// TwinCAT 3 PLC project PLC1
// ProgramVersion: 3.1.4026.16
// libraries:
//   Tc2_Standard, * (Beckhoff Automation GmbH)
//   Tc2_System, * (Beckhoff Automation GmbH)
// project tree:
//   DUTs/ YOLO_OBJECT_DETECTION.TcDUT
//   / PlcTask.TcTTO
//   POUs/ CountAndKeepValidDetections.TcPOU, MAIN.TcPOU, NonMaximumSuppression.TcPOU, SortDetectionsByConfidence.TcPOU
// real-time tasks:
//   TASK PlcTask: cycle T#10ms, priority 20, ADS port 350

CONFIGURATION PLC1
    RESOURCE PLC ON TwinCAT3
        TASK PlcTask(INTERVAL := T#10ms, PRIORITY := 20);
        PROGRAM MAIN WITH PlcTask : MAIN;
    END_RESOURCE
END_CONFIGURATION

// ---- DUTs/YOLO_OBJECT_DETECTION.TcDUT
TYPE YOLO_OBJECT_DETECTION :
STRUCT
	x_center_px 	: REAL;
    y_center_px 	: REAL;
    width_px    	: REAL;
    height_px   	: REAL;
    confidence  	: REAL;
	nTopLeftX       : REAL;
    nTopLeftY       : REAL;
    nBottomRightX   : REAL;
    nBottomRightY   : REAL;
    valid       	: BOOL; // For NMS marking
END_STRUCT
END_TYPE

// ---- POUs/MAIN.TcPOU
PROGRAM MAIN
VAR
	arrDetections : ARRAY[1..100] OF YOLO_OBJECT_DETECTION;
	numberOfDetections : INT := 100;
	numberOfValidDetections : INT ;
	bInit : BOOL;
END_VAR

IF NOT bInit THEN
	bInit := TRUE;
	arrDetections[1].nTopLeftX := 245;
	arrDetections[1].nTopLeftY := 305;
	arrDetections[1].nBottomRightX := 575;
	arrDetections[1].nBottomRightY := 490;	
	arrDetections[1].confidence := 0.2;
	arrDetections[1].valid := TRUE;
	arrDetections[2].nTopLeftX := 235;
	arrDetections[2].nTopLeftY := 300;
	arrDetections[2].nBottomRightX := 485;
	arrDetections[2].nBottomRightY := 515;	
	arrDetections[2].confidence := 0.3;
	arrDetections[2].valid := TRUE;	
	arrDetections[3].nTopLeftX := 305;
	arrDetections[3].nTopLeftY := 270;
	arrDetections[3].nBottomRightX := 540;
	arrDetections[3].nBottomRightY := 500;	
	arrDetections[3].confidence := 0.4;
	arrDetections[3].valid := TRUE;
	arrDetections[4].nTopLeftX := 800;
	arrDetections[4].nTopLeftY := 800;
	arrDetections[4].nBottomRightX := 1000;
	arrDetections[4].nBottomRightY := 1000;	
	arrDetections[4].confidence := 0.8;
	arrDetections[4].valid := TRUE;
END_IF

numberOfValidDetections := CountAndKeepValidDetections(detections:= ADR(arrDetections), count:= numberOfDetections);

IF numberOfValidDetections > 1 THEN
	IF SortDetectionsByConfidence(detections:= ADR(arrDetections), count:=numberOfValidDetections ) THEN
		NonMaximumSuppression(detections:= ADR(arrDetections), count:= numberOfValidDetections, iouThreshold:= 0.5);
	END_IF
END_IF

END_PROGRAM

// ---- POUs/CountAndKeepValidDetections.TcPOU
FUNCTION CountAndKeepValidDetections : INT
VAR_INPUT
	// Array containing 1 -- 100 predictions
    detections : POINTER TO ARRAY[1..100] OF YOLO_OBJECT_Detection; // Pointer to detection array
	// Number of valid non-valid predictions
    count : INT; // Original number of detections
END_VAR
VAR
	i : INT; // Current read index
    j : INT; // Write index for valid detections
END_VAR

j := 1; // Start writing at position 1

FOR i := 1 TO count DO
    IF detections^[i].valid THEN
        // Keep this detection
        IF i <> j THEN
            detections^[j] := detections^[i]; // Move valid detection forward
        END_IF
        j := j + 1;
    END_IF
END_FOR

// Optional: clear the rest of the array (not strictly necessary, but safe)
FOR i := j TO count DO
    detections^[i].valid := FALSE; // Mark remaining entries as invalid
END_FOR

CountAndKeepValidDetections := j - 1; // Return new count of valid detections

END_FUNCTION

// ---- POUs/SortDetectionsByConfidence.TcPOU
FUNCTION SortDetectionsByConfidence : BOOL
VAR_INPUT
	 detections : POINTER TO ARRAY[1..100] OF YOLO_OBJECT_DETECTION; // Pointer to array
    count : INT; // Number of valid detections
END_VAR
VAR
	i : INT;
    j : INT;
    temp : YOLO_OBJECT_DETECTION;
    swapped : BOOL;
END_VAR

SortDetectionsByConfidence := FALSE;

IF (count < 2) THEN
    RETURN; // Nothing to sort
END_IF

FOR i := 1 TO count - 1 DO
    swapped := FALSE;
    FOR j := 1 TO count - i DO
        // Sort by confidence descending
        IF detections^[j].confidence < detections^[j + 1].confidence THEN
            // Swap entire struct
            temp := detections^[j];
            detections^[j] := detections^[j + 1];
            detections^[j + 1] := temp;
            swapped := TRUE;
        END_IF
    END_FOR
    IF NOT swapped THEN
        EXIT;
    END_IF
END_FOR

SortDetectionsByConfidence := TRUE;

END_FUNCTION

// ---- POUs/NonMaximumSuppression.TcPOU
FUNCTION NonMaximumSuppression  : INT
VAR_INPUT
    detections : POINTER TO ARRAY[1..100] OF YOLO_OBJECT_Detection;
    count : INT; // Number of sorted detections (already sorted by confidence)
    iouThreshold : REAL; // Threshold to suppress, e.g., 0.5
END_VAR
VAR
	i, j : INT;
    iArea, jArea : REAL;
    xx1, yy1, xx2, yy2 : REAL;
    w, h : REAL;
    interArea, unionArea, iou : REAL;
    suppressedCount : INT := 0;
END_VAR

FOR i := 1 TO count DO
    IF NOT detections^[i].valid THEN
        CONTINUE; // Already suppressed
    END_IF

    iArea := (detections^[i].nBottomRightX - detections^[i].nTopLeftX) *
             (detections^[i].nBottomRightY - detections^[i].nTopLeftY);

    FOR j := i + 1 TO count DO
        IF NOT detections^[j].valid THEN
            CONTINUE;
        END_IF

        // Calculate intersection rectangle
        xx1 := MAX(detections^[i].nTopLeftX, detections^[j].nTopLeftX);
        yy1 := MAX(detections^[i].nTopLeftY, detections^[j].nTopLeftY);
        xx2 := MIN(detections^[i].nBottomRightX, detections^[j].nBottomRightX);
        yy2 := MIN(detections^[i].nBottomRightY, detections^[j].nBottomRightY);

        w := xx2 - xx1;
        h := yy2 - yy1;

        IF (w > 0.0) AND (h > 0.0) THEN
            interArea := w * h;

            jArea := (detections^[j].nBottomRightX - detections^[j].nTopLeftX) *
                     (detections^[j].nBottomRightY - detections^[j].nTopLeftY);

            unionArea := iArea + jArea - interArea;

            IF unionArea > 0.0 THEN
                iou := interArea / unionArea;

                IF iou > iouThreshold THEN
                    detections^[j].valid := FALSE; // Suppress overlapping detection
                    suppressedCount := suppressedCount + 1;
                END_IF
            END_IF
        END_IF
    END_FOR
END_FOR

NonMaximumSuppression := suppressedCount;

END_FUNCTION
